// TIA Portal project "encoder_jundiai" (V16)

(* hardware
DEVICE "S7-1200 station_1"  S7-1200 Station
   slot 0: "Rack_0"  S7-1200 Rack  Rack  V1.0
   slot 1: "PLC_1"  CPU 1211C AC/DC/Rly  6ES7 211-1BE40-0XB0  V4.4
*)

// ===== PLC "PLC_1"  CPU 1211C AC/DC/Rly =====

VAR_GLOBAL   // PLC tag table "Default tag table"
   "encoder_bk10_2201" AT %ID1000 : DInt;
   "ativar_motor_bk10_2201" AT %M0.0 : Bool;
   "ativar_motor_bk10_2201(1)" AT %Q0.0 : Bool;
   "aut/man_bk10_2201" AT %I0.2 : Bool;
   "encoder_branco_bk10_2201" AT %I0.0 : Bool;
   "sinaleiro _bk10_2201" AT %Q0.1 : Bool;
   "liga_motor_manual_bk10_2201" AT %I0.4 : Bool;
   "encoder_bk10_2301" AT %ID1004 : DInt;
   "ativar_motor_bk10_2301" AT %M0.1 : Bool;
   "ativar_motor_bk10_2301(1)" AT %Q0.2 : Bool;
   "aut/man_bk10_2301" AT %I0.3 : Bool;
   "encoder_branco_bk10_2301" AT %I0.1 : Bool;
   "sinaleiro _bk10_2301" AT %Q0.3 : Bool;
   "liga_motor_manual_bk10_2301" AT %I0.5 : Bool;
END_VAR

// folder: System blocks/Program resources

DATA_BLOCK "Timer_bk10_2201"   // DB2
{ S7_Optimized_Access := 'TRUE' }
AUTHOR : Simatic
FAMILY : IEC
NAME : IEC_TMR
VERSION : 1.0
// stored: InstanceOfName IEC_TIMER
"IEC_TIMER"
BEGIN
END_DATA_BLOCK

DATA_BLOCK "Timer_bk10_2301"   // DB4
{ S7_Optimized_Access := 'TRUE' }
AUTHOR : Simatic
FAMILY : IEC
NAME : IEC_TMR
VERSION : 1.0
// stored: InstanceOfName IEC_TIMER
"IEC_TIMER"
BEGIN
END_DATA_BLOCK

// folder: (top level)

ORGANIZATION_BLOCK "ob_bk10_2201"   // OB1, LAD, ProgramCycle
TITLE = "Main Program Sweep (Cycle)"
{ S7_Optimized_Access := 'TRUE' }
VERSION : 0.1
   VAR_INPUT
      Initial_Call : Bool;   // Initial call of this OB
      Remanence : Bool;   // =True, if remanent data are available
   END_VAR
BEGIN

REGION Network 1
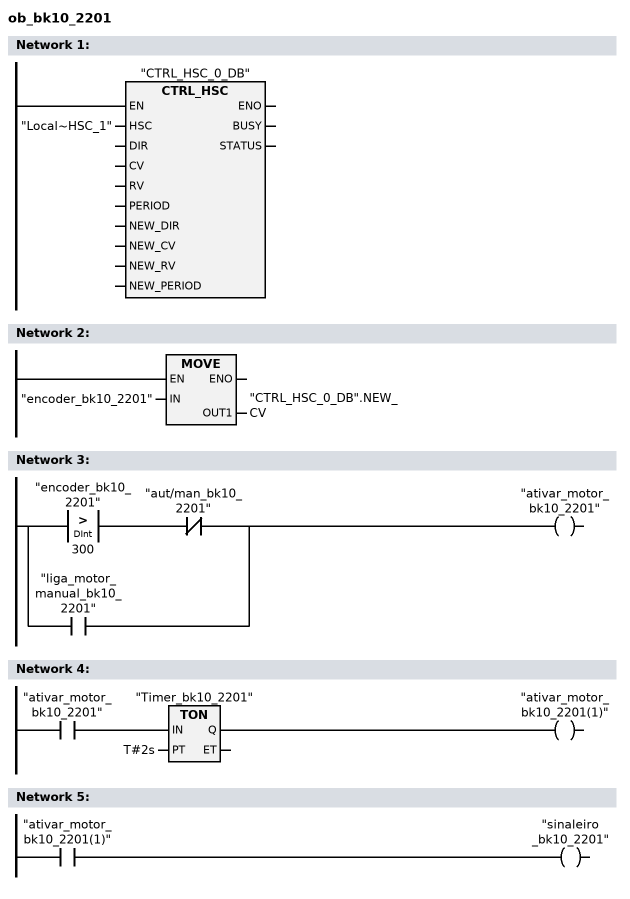
   "CTRL_HSC_0_DB"(HSC := "Local~HSC_1");   // CTRL_HSC
END_REGION

REGION Network 2
   RUNG wire#powerrail
      Move(in := "encoder_bk10_2201", out1 => "CTRL_HSC_0_DB".NEW_CV)
   END_RUNG
   // the same network as SCL:
   "CTRL_HSC_0_DB".NEW_CV := "encoder_bk10_2201";
END_REGION

REGION Network 3
   RUNG wire#powerrail
      { S7_Templates := "SrcType := DInt" } GT_Contact(in1 := "encoder_bk10_2201", in2 := 300)
      I_Contact( "aut/man_bk10_2201" )
      wire#w1
      Coil( "ativar_motor_bk10_2201" )
   END_RUNG
   RUNG wire#powerrail
      Contact( "liga_motor_manual_bk10_2201" )
   END_RUNG wire#w1
   // the same network as SCL:
   "ativar_motor_bk10_2201" := (("encoder_bk10_2201" > 300) AND NOT "aut/man_bk10_2201") OR "liga_motor_manual_bk10_2201";
END_REGION

REGION Network 4
   "Timer_bk10_2201".TON(IN := "ativar_motor_bk10_2201", PT := T#2s);
   "ativar_motor_bk10_2201(1)" := "Timer_bk10_2201".Q;
END_REGION

REGION Network 5
   RUNG wire#powerrail
      Contact( "ativar_motor_bk10_2201(1)" )
      Coil( "sinaleiro _bk10_2201" )
   END_RUNG
   // the same network as SCL:
   "sinaleiro _bk10_2201" := "ativar_motor_bk10_2201(1)";
END_REGION
END_ORGANIZATION_BLOCK

ORGANIZATION_BLOCK "ob_bk10_2301"   // OB123, LAD, ProgramCycle
TITLE = "Main Program Sweep (Cycle)"
{ S7_Optimized_Access := 'TRUE' }
VERSION : 0.1
   VAR_INPUT
      Initial_Call : Bool;   // Initial call of this OB
      Remanence : Bool;   // =True, if remanent data are available
   END_VAR
BEGIN

REGION Network 1
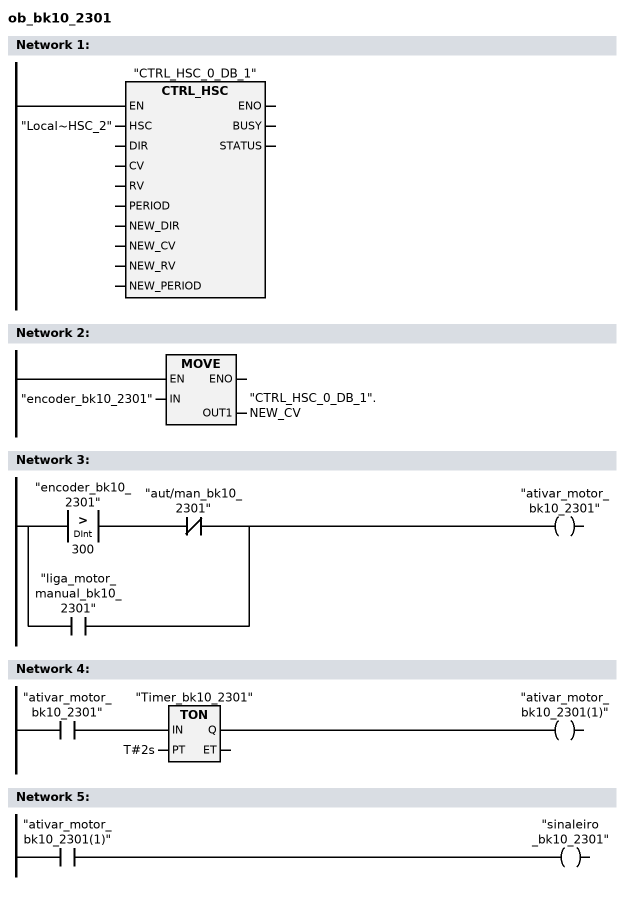
   "CTRL_HSC_0_DB_1"(HSC := "Local~HSC_2");   // CTRL_HSC
END_REGION

REGION Network 2
   RUNG wire#powerrail
      Move(in := "encoder_bk10_2301", out1 => "CTRL_HSC_0_DB_1".NEW_CV)
   END_RUNG
   // the same network as SCL:
   "CTRL_HSC_0_DB_1".NEW_CV := "encoder_bk10_2301";
END_REGION

REGION Network 3
   RUNG wire#powerrail
      { S7_Templates := "SrcType := DInt" } GT_Contact(in1 := "encoder_bk10_2301", in2 := 300)
      I_Contact( "aut/man_bk10_2301" )
      wire#w1
      Coil( "ativar_motor_bk10_2301" )
   END_RUNG
   RUNG wire#powerrail
      Contact( "liga_motor_manual_bk10_2301" )
   END_RUNG wire#w1
   // the same network as SCL:
   "ativar_motor_bk10_2301" := (("encoder_bk10_2301" > 300) AND NOT "aut/man_bk10_2301") OR "liga_motor_manual_bk10_2301";
END_REGION

REGION Network 4
   "Timer_bk10_2301".TON(IN := "ativar_motor_bk10_2301", PT := T#2s);
   "ativar_motor_bk10_2301(1)" := "Timer_bk10_2301".Q;
END_REGION

REGION Network 5
   RUNG wire#powerrail
      Contact( "ativar_motor_bk10_2301(1)" )
      Coil( "sinaleiro _bk10_2301" )
   END_RUNG
   // the same network as SCL:
   "sinaleiro _bk10_2301" := "ativar_motor_bk10_2301(1)";
END_REGION
END_ORGANIZATION_BLOCK